# EPICS StreamDevice protocol: GID/GID.proto
Terminator = CR LF;
ExtraInput = Ignore;
readGID {
	in "COM +%f ABN ABN NOR";
}
